// LS Electric XG5000 project: Project_RobotArm_PLC
// PLC LSPLC
// module base 0 slot 0: 입출력 모듈:XBC-DR32H (DC 24V 입력, 릴레이 출력 32점)

PROGRAM NewProgram (task: 스캔 프로그램)

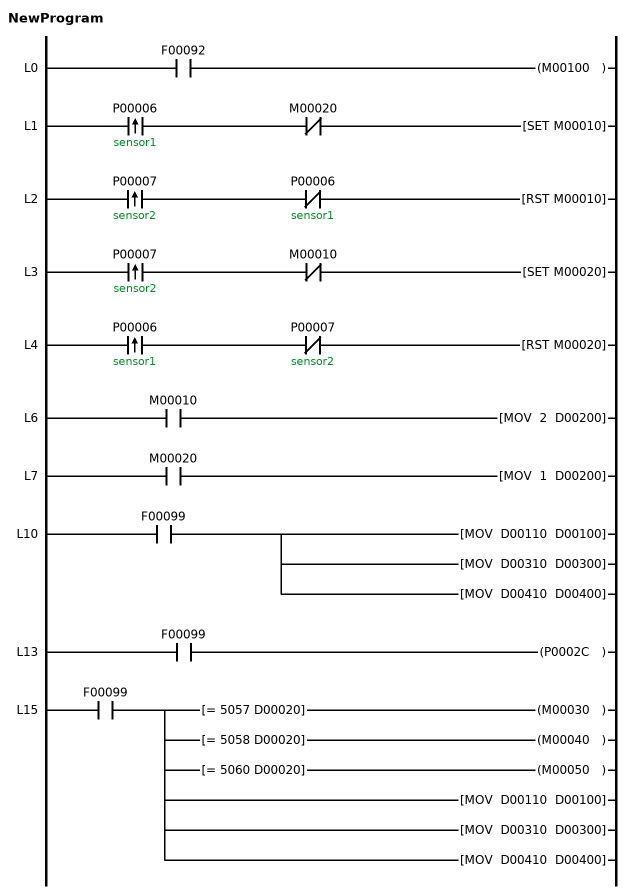
; L0
LOAD      F00092
OUT       M00100
; L1
LOADP     P00006	// sensor1
AND NOT   M00020
SET       M00010
; L2
LOADP     P00007	// sensor2
AND NOT   P00006	// sensor1
RST       M00010
; L3
LOADP     P00007	// sensor2
AND NOT   M00010
SET       M00020
; L4
LOADP     P00006	// sensor1
AND NOT   P00007	// sensor2
RST       M00020
; L6
LOAD      M00010
MOV       2 D00200
; L7
LOAD      M00020
MOV       1 D00200
; L10
LOAD      F00099
MOV       D00110 D00100
MOV       D00310 D00300
MOV       D00410 D00400
; L13
LOAD      F00099
OUT       P0002C
; L15
LOAD      F00099
MPUSH
AND=      5057 D00020
OUT       M00030
MLOAD
AND=      5058 D00020
OUT       M00040
MLOAD
AND=      5060 D00020
OUT       M00050
MPOP
MOV       D00110 D00100
MOV       D00310 D00300
MOV       D00410 D00400

VARIABLES AND COMMENTS (devices not used above)
P00001	BIT	PB1
P00002	BIT	PB2